INTERFACE I_ListNode EXTENDS I_CollectionNode;

END_INTERFACE

(* stored: Version 1.1.0.1, ProductVersion 3.1.4024.12
   Itf I_ListNode: Id {92604193-4296-06cc-11b0-8b3359e8272f} *)
